Universal Robots PolyScope program: gripper_close.urp

Program gripper_close (installation=default directory=/programs/usbdisk createdIn=5.12.6.1102099 lastSavedIn=5.12.6.1102099 robotSerialNumber=20195001816)
Calibrated DH parameters: a=[0.000205, -0.596127, -0.182301, -0.000015, 0.000015, 0]; d=[0.180703, -32.967112, 471.012495, -437.871095, 0.119874, 0.115473]; alpha=[1.570442, -0.004218, 0.001236, 1.571679, -1.571534, 0]; deltaTheta=[0, 0.229143, 7.300074, -1.246036, -0.000003, 0]
Robot Program (runOnlyOnce=false)
  URCap Gripper (Robotiq_Grippers, Robotiq Inc.) dataModel(position=100.0, force=80.0, speed=80.0, positionInDouble=100.0, forceInDouble=80.0, speedInDouble=80.0, slaveIds=[9], blocking=true)
